// Mitsubishi GX Works2 project: SET_RST   PLC: Q03UDV

PROGRAM MAIN
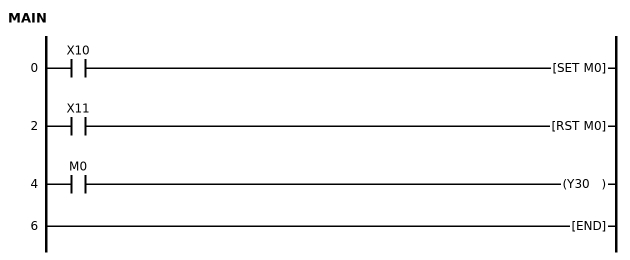
0     LD      X10
      SET     M0
2     LD      X11
      RST     M0
4     LD      M0
      OUT     Y30
6     END
END_PROGRAM
